(*	HMI variables

	This block holds all HMI variables and handles communication with the HMI
	
	2024-02 HP
		-initial
*)

{attribute 'no_explicit_call' := 'do not call this POU directly'}
FUNCTION_BLOCK HMI_SafetyGroup1 EXTENDS HMI_BaseBlock
//HMI variables that can be written to by the plc and HMI 
VAR_INPUT
	//Do not change these names, the HMI is hardcoded to use these exact names
	MAN:HMI_NotUsed;				//HMI manuals
	STS:HMI_STS_SafetyGroup1;		//HMI statusses
	WRN:HMI_WRN_SafetyGroup1;		//HMI warnings
	ERR:HMI_ERR_SafetyGroup1;		//HMI errors
END_VAR

//Hmi variables that can only be written to by the HMI and read by the plc
VAR_OUTPUT PERSISTENT
	//Do not change these names, the HMI is hardcoded to use these exact names
	//SP:HMI_SP_SafetyLogic;			//HMI setpoints
END_VAR

//this block should not be called

END_FUNCTION_BLOCK

(* stored: Version 1.1.0.1
   POU HMI_SafetyGroup1: Id {8fee68d7-3918-0caf-3a4e-836782cbe436}, SpecialFunc None *)
